{attribute 'linkalways'} 
{attribute 'no_explicit_call' := 'This FB is a CLASS and must be accessed using methods or properties'}
{attribute 'enable_dynamic_creation'}
FUNCTION_BLOCK FINAL MOD_DINT EXTENDS Node
VAR
	in1 : _DINT(0);
	in2 : _DINT(0);
	out : _DINT(0);
END_VAR

METHOD PUBLIC Clone : I_Node
VAR
	pNode : POINTER TO MOD_DINT;
END_VAR
pNode := __NEW(MOD_DINT);
Clone := pNode^;
END_METHOD

METHOD FB_init : BOOL
VAR_INPUT
	bInitRetains : BOOL; // if TRUE, the retain variables are initialized (warm start / cold start)
	bInCopyCode : BOOL;  // if TRUE, the instance afterwards gets moved into the copy code (online change)
END_VAR
AddInput('in1',THIS^.in1);
AddInput('in2',THIS^.in2);
AddOutput('out', THIS^.out);
END_METHOD

METHOD PROTECTED OnExecute
VAR
END_VAR
out.Value := in1.Value MOD in2.Value;
END_METHOD

END_FUNCTION_BLOCK

(* stored: Version 1.1.0.1, ProductVersion 3.1.4024.15
   POU MOD_DINT: Id {40f9b367-fbf3-4a4c-a81a-ce3b0c228bd7}, SpecialFunc None
   Folder Constructor: Id {80491308-3d50-4dbc-8c43-637327ede43c}
   Method Clone: Id {db4ecaf4-36b4-42e3-873b-dbdb6b9490b9}
   Method FB_init: Id {6e57b0f8-b35d-4ef6-89b2-59b3ea68afd3}
   Method OnExecute: Id {8e02a02e-14f5-4bff-a671-335ec7bd6eef} *)
